FUNCTION_BLOCK FB_HYST_1 (* Basic Function Block Type *)
  (* Standard: 61499-2 *)
  (* Version 0.0, 2011-08-31, 4DIAC-IDE, 4DIAC-Consortium *)
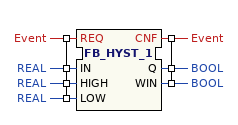
  EVENT_INPUT
    REQ WITH IN, HIGH, LOW; (* Normal Execution Request *)
  END_EVENT
  EVENT_OUTPUT
    CNF WITH WIN, Q; (* Execution Confirmation *)
  END_EVENT
  VAR_INPUT
    IN : REAL; (* input value *)
    HIGH : REAL; (* upper threshold *)
    LOW : REAL; (* lower threshold *)
  END_VAR
  VAR_OUTPUT
    Q : BOOL; (* output *)
    WIN : BOOL; (* shows that IN lies in between HIGH and LOW *)
  END_VAR
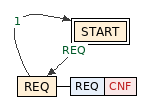
  EC_STATES
    START; (* Initial State *)
    REQ : REQ -> CNF; (* Normal execution *)
  END_STATES
  EC_TRANSITIONS
    START TO REQ := REQ;
    REQ TO START := 1;
  END_TRANSITIONS
  ALGORITHM REQ IN ST: (* Normally executed algorithm *)
IF IN < LOW THEN
	Q := FALSE;
	WIN := FALSE;
ELSIF IN > HIGH THEN
	Q := TRUE;
	WIN := FALSE;
ELSE
	WIN := TRUE;
END_IF;
  END_ALGORITHM
END_FUNCTION_BLOCK
